FUNCTION ANLG_TO_ABC : LREAL
VAR_INPUT
	iMn : REAL;
	iMx : REAL;
	oMn : REAL;
	oMx : REAL;
	ofs : REAL := 0; //offset
	val : DINT;
	b: REAL :=0.0;
END_VAR
VAR
	temp:LREAL;
END_VAR

temp:= SEL(b=0.0,
	   ((oMx-oMn)/(iMx-iMn))*val + b,  
	   ((oMx-oMn)/(iMx-iMn))*val + (oMn -((oMx-oMn)/(iMx-iMn))*iMn));
				 
				 
ANLG_TO_ABC:=SEL(temp<ofs AND ofs<>0 AND oMn=0, temp+ofs, temp); 				 
				 			 
(*				 
ANLG_TO_ABC:= SEL(b=0.0,
				 ((oMx-oMn)/(iMx-iMn))*val + ofs + b,  
				 ((oMx-oMn)/(iMx-iMn))*val + ofs + (oMn -((oMx-oMn)/(iMx-iMn))*iMn));	
*)

END_FUNCTION

(* stored: Version 1.1.0.1, ProductVersion 3.1.4022.18
   POU ANLG_TO_ABC: Id {bbe9b7ab-1d84-4de0-b840-2ec1f6c9fa5f}, SpecialFunc None *)
